Staubli VAL3: PriseEnMain.pjx

--- PriseEnMain.pjx ---
Parameters version=s8.10.3Cs9_BS2093 stackSize=5000 millimeterUnit=true
Program file=Deplacement.pgx
Program file=IO.pgx
Program file=start.pgx
Program file=stop.pgx
Program file=Variables.pgx
Data file=PriseEnMain.dtx

--- PriseEnMain.dtx ---
mdesc mNomSpeed
jointRx jInit
jointRx jDest
pointRx pCarre1 = {fatherId=world[0]}
pointRx pCarre2 = {fatherId=world[0]}
pointRx pCarre4 = {fatherId=world[0]}
pointRx pCarre3 = {fatherId=world[0]}

--- start.pgx ---
program start()
begin
  call Variables()
  call IO()
  call Deplacement()
end

--- Deplacement.pgx ---
program Deplacement()
begin
  movej(jInit, flange, mNomSpeed)
  movej(jDest, flange, mNomSpeed)
  waitEndMove()

  do
    waitEndMove()
    //movel(pCarre1, flange, mNomSpeed)
    //movel(pCarre2, flange, mNomSpeed)
    movec(pCarre1, pCarre2, flange, mNomSpeed)
    movej(pCarre3, flange, mNomSpeed)
    movej(pCarre4, flange, mNomSpeed)
  until false
end

--- IO.pgx ---
program IO()
begin
end

--- Variables.pgx ---
program Variables()
begin
  jInit = {0,0,0,0,0,0}
  jDest = {0,90,-90,0,0,0}
  pCarre1 = {{0,600,500,0,0,0}, {sfree, efree, wfree}}
  pCarre2 = {{-500,0,500,0,0,0}, {sfree, efree, wfree}}
  pCarre3 = {{0,-500,500,0,0,0}, {sfree, efree, wfree}}
  pCarre4 = {{500,0,500,0,0,0}, {sfree, efree, wfree}}
end
